VAR_GLOBAL
	// NOTE: Following parameters are bogus, make sure to add real ones...
	// M1L0
	M1L0_Pitch	    :	HOMS_PitchMechanism := (
		ReqPosLimHi := 21850,
		ReqPosLimLo := 14800,
		diEncPosLimHi := 11256000,
		diEncPosLimLo := 7561000
	);

	{attribute 'TcLinkTo' := '.bLimitForwardEnable:=TIIB[EL7041-1000_M2L0_PitchCoarse]^STM Status^Status^Digital input 1;
                              .bLimitBackwardEnable:=TIIB[EL7041-1000_M2L0_PitchCoarse]^STM Status^Status^Digital input 2'}
	{attribute 'pytmc' := '
		pv: MR2L0:LFE:MMS:PITCH
	'}
	M11 : DUT_MotionStage:=(nEnableMode:=ENUM_StageEnableMode.STAGE_ENABLE_MOTION,
                            nCommand:=ENUM_EpicsMotorCmd.EPICS_MOTOR_MOVE_ABS); // PitchCoarse
	// M2L0
	M2L0_Pitch	    :	HOMS_PitchMechanism := (
		Stepper := M11,
		ReqPosLimHi := 20000,
		ReqPosLimLo := 16500,
		diEncPosLimHi := 10722213,
		diEncPosLimLo := 8208000
	);
END_VAR

(* stored: Version 1.1.0.1, ProductVersion 3.1.4022.12
   GVL GVL_Devices: Id {cb7cf638-cc80-4f58-a532-470704faedf8} *)
